// TwinCAT 3 PLC project BottleFillingLine
// ProgramVersion: 3.1.4024.0
// libraries:
//   Tc2_Standard, * (Beckhoff Automation GmbH)
//   Tc2_System, * (Beckhoff Automation GmbH)
//   Tc3_Module, * (Beckhoff Automation GmbH)
// project tree:
//   / E_PackMLState.TcDUT, FB_UnitStateMachine.TcPOU, PlcTask.TcTTO
//   GVLs/ GVL_PackML.TcGVL
//   POUs/ FB_CappingStation.TcPOU, FB_FillStation.TcPOU, FB_InfeedConveyor.TcPOU, MAIN.TcPOU
// real-time tasks:
//   TASK PlcTask: cycle T#10ms, priority 20, ADS port 350

CONFIGURATION BottleFillingLine
    RESOURCE PLC ON TwinCAT3
        TASK PlcTask(INTERVAL := T#10ms, PRIORITY := 20);
        PROGRAM MAIN WITH PlcTask : MAIN;
    END_RESOURCE
END_CONFIGURATION

// ---- E_PackMLState.TcDUT
{attribute 'qualified_only'}
TYPE E_PackMLState :
(
    Undefined    := 0,
    Clearing     := 1,
    Stopped      := 2,
    Starting     := 3,
    Idle         := 4,
    Suspended    := 5,
    Execute      := 6,
    Stopping     := 7,
    Aborting     := 8,
    Aborted      := 9,
    Holding      := 10,
    Held         := 11,
    Unholding    := 12,
    Suspending   := 13,
    Unsuspending := 14,
    Resetting    := 15,
    Completing   := 16,
    Complete     := 17
);
END_TYPE

// ---- GVLs/GVL_PackML.TcGVL
{attribute 'qualified_only'}
VAR_GLOBAL
    // Unit state machine status
    UnitCurrentState    : E_PackMLState;    // Mirror of UnitSM.CurrentState

    // Infeed conveyor
    InfeedBottleCount   : INT;              // Total bottles entering the line

    // Fill station
    FillLevel           : REAL;             // Current fill level 0.0 - 100.0

    // Capping station
    CapsApplied         : INT;              // Total caps applied
END_VAR

// ---- POUs/MAIN.TcPOU
PROGRAM MAIN
VAR
    // Unit state machine
    UnitSM         : FB_UnitStateMachine;

    // Station function blocks — instantiated here, called every scan
    Infeed         : FB_InfeedConveyor;
    FillStn        : FB_FillStation;
    CappingStn     : FB_CappingStation;

    // Operator command buttons — toggle manually in the watch window
    cmd_Reset      : BOOL;
    cmd_Start      : BOOL;
    cmd_Stop       : BOOL;
    cmd_Hold       : BOOL;
    cmd_UnHold     : BOOL;
    cmd_Suspend    : BOOL;
    cmd_UnSuspend  : BOOL;
    cmd_Abort      : BOOL;
    cmd_Clear      : BOOL;
END_VAR

// ── Unit State Machine ────────────────────────────────────────────────────────
// Call every scan cycle, pass operator commands in
// The FB handles all state logic internally
UnitSM(
    SC_Reset      := cmd_Reset,
    SC_Start      := cmd_Start,
    SC_Stop       := cmd_Stop,
    SC_Hold       := cmd_Hold,
    SC_UnHold     := cmd_UnHold,
    SC_Suspend    := cmd_Suspend,
    SC_UnSuspend  := cmd_UnSuspend,
    SC_Abort      := cmd_Abort,
    SC_Clear      := cmd_Clear
);

// Auto-clear commands after one scan so they act as pulses not holds
// This mimics a real momentary button press
cmd_Reset     := FALSE;
cmd_Start     := FALSE;
cmd_Stop      := FALSE;
cmd_Hold      := FALSE;
cmd_UnHold    := FALSE;
cmd_Suspend   := FALSE;
cmd_UnSuspend := FALSE;
cmd_Abort     := FALSE;
cmd_Clear     := FALSE;

// ── Station Function Blocks ───────────────────────────────────────────────────
// Called every scan, each station drives itself based on unit state
Infeed(
    UnitState := UnitSM.CurrentState
);

FillStn(
    UnitState := UnitSM.CurrentState
);

CappingStn(
    UnitState := UnitSM.CurrentState
);

// ── GVL Mirror ────────────────────────────────────────────────────────────────
// Copy station outputs to global dashboard every scan
// Anything in the program can now read these without touching the FBs directly
GVL_PackML.UnitCurrentState  := UnitSM.CurrentState;
GVL_PackML.InfeedBottleCount := Infeed.BottleCount;
GVL_PackML.FillLevel         := FillStn.FillLevel;
GVL_PackML.CapsApplied       := CappingStn.CapsApplied;

END_PROGRAM

// ---- FB_UnitStateMachine.TcPOU
FUNCTION_BLOCK FB_UnitStateMachine
VAR_INPUT
    // Commands from operator or supervisor — these are the SC_ signals in PackML
    SC_Reset      : BOOL;  // Stopped → Resetting
    SC_Start      : BOOL;  // Idle → Starting
    SC_Stop       : BOOL;  // Any state → Stopping
    SC_Hold       : BOOL;  // Execute → Holding
    SC_UnHold     : BOOL;  // Held → Unholding
    SC_Suspend    : BOOL;  // Execute → Suspending
    SC_UnSuspend  : BOOL;  // Suspended → Unsuspending
    SC_Abort      : BOOL;  // Any state → Aborting
    SC_Clear      : BOOL;  // Aborted → Clearing
END_VAR

VAR_OUTPUT
    // Current state readable by anything outside this FB
    CurrentState  : E_PackMLState;
END_VAR

VAR
    // Internal timer — acting states use this to simulate work taking time
    StateTimer    : TON;
END_VAR

// PackML Unit State Machine
// Runs every PLC scan cycle — checks current state and transitions if conditions are met

// SC_Abort is valid from ANY state — highest priority check
IF SC_Abort THEN
    CurrentState := E_PackMLState.Aborting;
END_IF

CASE CurrentState OF

    E_PackMLState.Undefined:
        // Starting point — immediately go to Stopped on first scan
        CurrentState := E_PackMLState.Stopped;

    E_PackMLState.Stopped:
        // Stable state — wait here until SC_Reset received
        IF SC_Reset THEN
            CurrentState := E_PackMLState.Resetting;
        END_IF

    E_PackMLState.Resetting:
        // Acting state — simulate hardware init with a 2 second timer
        StateTimer(IN := TRUE, PT := T#2S);
        IF StateTimer.Q THEN
            StateTimer(IN := FALSE);  // Reset timer
            CurrentState := E_PackMLState.Idle;
        END_IF

    E_PackMLState.Idle:
        // Stable state — machine ready, wait for SC_Start
        IF SC_Start THEN
            CurrentState := E_PackMLState.Starting;
        END_IF

    E_PackMLState.Starting:
        // Acting state — simulate startup sequence with a 1 second timer
        StateTimer(IN := TRUE, PT := T#1S);
        IF StateTimer.Q THEN
            StateTimer(IN := FALSE);
            CurrentState := E_PackMLState.Execute;
        END_IF

    E_PackMLState.Execute:
        // Stable state — production running
        IF SC_Hold THEN
            CurrentState := E_PackMLState.Holding;
        ELSIF SC_Suspend THEN
            CurrentState := E_PackMLState.Suspending;
        ELSIF SC_Stop THEN
            CurrentState := E_PackMLState.Stopping;
        END_IF

    E_PackMLState.Holding:
        // Acting state — controlled pause sequence
        StateTimer(IN := TRUE, PT := T#1S);
        IF StateTimer.Q THEN
            StateTimer(IN := FALSE);
            CurrentState := E_PackMLState.Held;
        END_IF

    E_PackMLState.Held:
        // Stable state — paused, wait for SC_UnHold
        IF SC_UnHold THEN
            CurrentState := E_PackMLState.Unholding;
        END_IF

    E_PackMLState.Unholding:
        // Acting state — resume from hold
        StateTimer(IN := TRUE, PT := T#1S);
        IF StateTimer.Q THEN
            StateTimer(IN := FALSE);
            CurrentState := E_PackMLState.Execute;
        END_IF

    E_PackMLState.Suspending:
        // Acting state — entering suspended
        StateTimer(IN := TRUE, PT := T#1S);
        IF StateTimer.Q THEN
            StateTimer(IN := FALSE);
            CurrentState := E_PackMLState.Suspended;
        END_IF

    E_PackMLState.Suspended:
        // Stable state — starved or blocked, wait for SC_UnSuspend
        IF SC_UnSuspend THEN
            CurrentState := E_PackMLState.Unsuspending;
        END_IF

    E_PackMLState.Unsuspending:
        // Acting state — resuming from suspended
        StateTimer(IN := TRUE, PT := T#1S);
        IF StateTimer.Q THEN
            StateTimer(IN := FALSE);
            CurrentState := E_PackMLState.Execute;
        END_IF

    E_PackMLState.Stopping:
        // Acting state — controlled stop sequence
        StateTimer(IN := TRUE, PT := T#2S);
        IF StateTimer.Q THEN
            StateTimer(IN := FALSE);
            CurrentState := E_PackMLState.Stopped;
        END_IF

    E_PackMLState.Aborting:
        // Acting state — emergency shutdown, gets here from any state
        StateTimer(IN := TRUE, PT := T#1S);
        IF StateTimer.Q THEN
            StateTimer(IN := FALSE);
            CurrentState := E_PackMLState.Aborted;
        END_IF

    E_PackMLState.Aborted:
        // Stable state — fault state, wait for SC_Clear
        IF SC_Clear THEN
            CurrentState := E_PackMLState.Clearing;
        END_IF

    E_PackMLState.Clearing:
        // Acting state — clear the fault
        StateTimer(IN := TRUE, PT := T#2S);
        IF StateTimer.Q THEN
            StateTimer(IN := FALSE);
            CurrentState := E_PackMLState.Stopped;
        END_IF

    E_PackMLState.Completing:
        // Acting state — end of batch wrap-up
        StateTimer(IN := TRUE, PT := T#2S);
        IF StateTimer.Q THEN
            StateTimer(IN := FALSE);
            CurrentState := E_PackMLState.Complete;
        END_IF

    E_PackMLState.Complete:
        // Stable state — batch done, await SC_Reset to run again
        IF SC_Reset THEN
            CurrentState := E_PackMLState.Resetting;
        END_IF

END_CASE

END_FUNCTION_BLOCK

// ---- POUs/FB_InfeedConveyor.TcPOU
FUNCTION_BLOCK FB_InfeedConveyor
VAR_INPUT
    // Commands passed down from the unit state machine
    Start         : BOOL;   // Unit entered Execute — start conveyor
    Stop          : BOOL;   // Unit stopping — stop conveyor
    Hold          : BOOL;   // Unit holding — pause conveyor
    Abort         : BOOL;   // Unit aborting — kill conveyor immediately
    UnitState     : E_PackMLState;    // Added: wired from UnitSM.CurrentState in MAIN
END_VAR

VAR_OUTPUT
    // Status reported up to the unit state machine
    Ready         : BOOL;   // TRUE when conveyor is running and ready
    Faulted       : BOOL;   // TRUE if a fault condition exists
    CurrentState  : E_PackMLState;
	BottleCount   : INT;    // Simulates bottles on the conveyor
END_VAR

VAR
    StateTimer    : TON;    // Simulates conveyor ramp-up and ramp-down time
END_VAR

// Infeed Conveyor Module State Machine
// Receives commands from unit, reports status back up

// Abort overrides everything — immediate stop
IF Abort THEN
    CurrentState  := E_PackMLState.Aborting;
    Ready         := FALSE;
END_IF

CASE CurrentState OF

    E_PackMLState.Undefined:
        // First scan — go to stopped
        CurrentState := E_PackMLState.Stopped;
        Ready        := FALSE;

    E_PackMLState.Stopped:
        Ready := FALSE;
        IF Start THEN
            CurrentState := E_PackMLState.Starting;
        END_IF

    E_PackMLState.Starting:
        // Simulate conveyor belt spinning up — 1.5 second ramp
        Ready := FALSE;
        StateTimer(IN := TRUE, PT := T#1500MS);
        IF StateTimer.Q THEN
            StateTimer(IN := FALSE);
            BottleCount  := 0;
            CurrentState := E_PackMLState.Execute;
        END_IF

    E_PackMLState.Execute:
        // Conveyor running — increment bottle count to simulate flow
        Ready       := TRUE;
        BottleCount := BottleCount + 1;
        IF Hold THEN
            CurrentState := E_PackMLState.Holding;
        ELSIF Stop THEN
            CurrentState := E_PackMLState.Stopping;
        END_IF

    E_PackMLState.Holding:
        // Controlled pause — conveyor slows down over 1 second
        Ready := FALSE;
        StateTimer(IN := TRUE, PT := T#1S);
        IF StateTimer.Q THEN
            StateTimer(IN := FALSE);
            CurrentState := E_PackMLState.Held;
        END_IF

    E_PackMLState.Held:
        // Paused — waiting for unit to send resume
        Ready := FALSE;
        IF Start THEN
            CurrentState := E_PackMLState.Unholding;
        END_IF

    E_PackMLState.Unholding:
        // Resuming from hold
        StateTimer(IN := TRUE, PT := T#1S);
        IF StateTimer.Q THEN
            StateTimer(IN := FALSE);
            CurrentState := E_PackMLState.Execute;
        END_IF

    E_PackMLState.Stopping:
        // Controlled stop — conveyor ramps down over 2 seconds
        Ready := FALSE;
        StateTimer(IN := TRUE, PT := T#2S);
        IF StateTimer.Q THEN
            StateTimer(IN := FALSE);
            CurrentState := E_PackMLState.Stopped;
        END_IF

    E_PackMLState.Aborting:
        // Immediate stop — no ramp down
        Ready  := FALSE;
        StateTimer(IN := TRUE, PT := T#500MS);
        IF StateTimer.Q THEN
            StateTimer(IN := FALSE);
            Faulted      := TRUE;
            CurrentState := E_PackMLState.Aborted;
        END_IF

    E_PackMLState.Aborted:
        // Fault state — waits for unit to clear
        Ready   := FALSE;
        Faulted := TRUE;

END_CASE

END_FUNCTION_BLOCK

// ---- POUs/FB_FillStation.TcPOU
FUNCTION_BLOCK FB_FillStation
VAR_INPUT
    Start         : BOOL;
    Stop          : BOOL;
    Hold          : BOOL;
    Abort         : BOOL;
	UnitState     : E_PackMLState;    // Added: wired from UnitSM.CurrentState in MAIN
END_VAR

VAR_OUTPUT
    Ready         : BOOL;
    Faulted       : BOOL;
    CurrentState  : E_PackMLState;
	FillLevel     : REAL;   // Simulates liquid fill level 0.0 to 100.0
END_VAR

VAR
    StateTimer    : TON;
END_VAR

// Fill Station Module State Machine
// Simulates a liquid fill valve opening and filling bottles

IF Abort THEN
    CurrentState := E_PackMLState.Aborting;
    Ready        := FALSE;
END_IF

CASE CurrentState OF

    E_PackMLState.Undefined:
        CurrentState := E_PackMLState.Stopped;
        Ready        := FALSE;

    E_PackMLState.Stopped:
        Ready     := FALSE;
        FillLevel := 0.0;
        IF Start THEN
            CurrentState := E_PackMLState.Starting;
        END_IF

    E_PackMLState.Starting:
        // Simulate valve priming — 2 second startup
        Ready := FALSE;
        StateTimer(IN := TRUE, PT := T#2S);
        IF StateTimer.Q THEN
            StateTimer(IN := FALSE);
            CurrentState := E_PackMLState.Execute;
        END_IF

    E_PackMLState.Execute:
        // Simulate fill level rising each scan
        Ready     := TRUE;
        FillLevel := FillLevel + 0.5;
        IF FillLevel >= 100.0 THEN
            FillLevel := 0.0;   // Reset for next bottle
        END_IF
        IF Hold THEN
            CurrentState := E_PackMLState.Holding;
        ELSIF Stop THEN
            CurrentState := E_PackMLState.Stopping;
        END_IF

    E_PackMLState.Holding:
        Ready := FALSE;
        StateTimer(IN := TRUE, PT := T#1S);
        IF StateTimer.Q THEN
            StateTimer(IN := FALSE);
            CurrentState := E_PackMLState.Held;
        END_IF

    E_PackMLState.Held:
        Ready := FALSE;
        IF Start THEN
            CurrentState := E_PackMLState.Unholding;
        END_IF

    E_PackMLState.Unholding:
        StateTimer(IN := TRUE, PT := T#1S);
        IF StateTimer.Q THEN
            StateTimer(IN := FALSE);
            CurrentState := E_PackMLState.Execute;
        END_IF

    E_PackMLState.Stopping:
        Ready     := FALSE;
        FillLevel := 0.0;
        StateTimer(IN := TRUE, PT := T#2S);
        IF StateTimer.Q THEN
            StateTimer(IN := FALSE);
            CurrentState := E_PackMLState.Stopped;
        END_IF

    E_PackMLState.Aborting:
        Ready := FALSE;
        StateTimer(IN := TRUE, PT := T#500MS);
        IF StateTimer.Q THEN
            StateTimer(IN := FALSE);
            Faulted      := TRUE;
            CurrentState := E_PackMLState.Aborted;
        END_IF

    E_PackMLState.Aborted:
        Ready   := FALSE;
        Faulted := TRUE;

END_CASE

END_FUNCTION_BLOCK

// ---- POUs/FB_CappingStation.TcPOU
FUNCTION_BLOCK FB_CappingStation
VAR_INPUT
    Start         : BOOL;
    Stop          : BOOL;
    Hold          : BOOL;
    Abort         : BOOL;
	UnitState     : E_PackMLState;    // Added: wired from UnitSM.CurrentState in MAIN
END_VAR

VAR_OUTPUT
    Ready         : BOOL;
    Faulted       : BOOL;
    CurrentState  : E_PackMLState;
	CapsApplied   : INT;    // Simulates cap count
END_VAR

VAR
    StateTimer    : TON;
END_VAR

// Capping Station Module State Machine
// Simulates a capping head applying caps to filled bottles

IF Abort THEN
    CurrentState := E_PackMLState.Aborting;
    Ready        := FALSE;
END_IF

CASE CurrentState OF

    E_PackMLState.Undefined:
        CurrentState := E_PackMLState.Stopped;
        Ready        := FALSE;

    E_PackMLState.Stopped:
        Ready       := FALSE;
        CapsApplied := 0;
        IF Start THEN
            CurrentState := E_PackMLState.Starting;
        END_IF

    E_PackMLState.Starting:
        // Simulate capping head homing — 1 second
        Ready := FALSE;
        StateTimer(IN := TRUE, PT := T#1S);
        IF StateTimer.Q THEN
            StateTimer(IN := FALSE);
            CurrentState := E_PackMLState.Execute;
        END_IF

    E_PackMLState.Execute:
        // Apply caps and count them
        Ready       := TRUE;
        CapsApplied := CapsApplied + 1;
        IF Hold THEN
            CurrentState := E_PackMLState.Holding;
        ELSIF Stop THEN
            CurrentState := E_PackMLState.Stopping;
        END_IF

    E_PackMLState.Holding:
        Ready := FALSE;
        StateTimer(IN := TRUE, PT := T#1S);
        IF StateTimer.Q THEN
            StateTimer(IN := FALSE);
            CurrentState := E_PackMLState.Held;
        END_IF

    E_PackMLState.Held:
        Ready := FALSE;
        IF Start THEN
            CurrentState := E_PackMLState.Unholding;
        END_IF

    E_PackMLState.Unholding:
        StateTimer(IN := TRUE, PT := T#1S);
        IF StateTimer.Q THEN
            StateTimer(IN := FALSE);
            CurrentState := E_PackMLState.Execute;
        END_IF

    E_PackMLState.Stopping:
        Ready := FALSE;
        StateTimer(IN := TRUE, PT := T#2S);
        IF StateTimer.Q THEN
            StateTimer(IN := FALSE);
            CurrentState := E_PackMLState.Stopped;
        END_IF

    E_PackMLState.Aborting:
        Ready := FALSE;
        StateTimer(IN := TRUE, PT := T#500MS);
        IF StateTimer.Q THEN
            StateTimer(IN := FALSE);
            Faulted      := TRUE;
            CurrentState := E_PackMLState.Aborted;
        END_IF

    E_PackMLState.Aborted:
        Ready   := FALSE;
        Faulted := TRUE;

END_CASE

END_FUNCTION_BLOCK
